// TIA Portal V21 export
FUNCTION_BLOCK "FB608"   // FB608, LAD
TITLE = FB608
{ S7_Optimized_Access := 'FALSE' }
AUTHOR : PRECISE
FAMILY : PRECISE
// CIP RECIRCULATION
// stored: AutoNumber false, SetENOAutomatically false
   VAR_INPUT
      CycleEnable : Bool;
      CycleRunning : Bool;
      SecPulse : Bool;
      AlwaysTrue : Bool;
      ActualTemperature : Real;
      ParaIn : "RecirculationInputs";
      ActualPressure : Real;
      ActualConductivity : Real;
   END_VAR
   VAR_OUTPUT
      Started : Bool;
      PressureUtilityValve : Bool;   // Air Utility
      AlkaliInValve : Bool;
      AlkaliPump : Bool;
      AcidInValve : Bool;
      AcidPump : Bool;
      "DosingValve(Cond)" : Bool;
      "DosingPump(Cond)" : Bool;
      HsbCmd : Bool;
      RecPump : Bool;
      ParaOut : "RecirculationOutputs";
      TimePv : DInt;
      StepStatus : String[60];
   END_VAR
   VAR_IN_OUT
      Over : Bool;
      OverTemp : Bool;
      ControlStarted : Bool;
      TimerPaused : Bool;
      PressurePostiveTol : Real;
      PressureNegativeTol : Real;
      LineValves : Bool;
      ActualRepetition : Int;
      SetTemperature { ExternalAccessible := 'False'; ExternalVisible := 'False'; ExternalWritable := 'False'} : Real;
      SetpH : Real;
      SetConductivity : Real;
      pHReached : Bool;
      ConductivityReached : Bool;
      CipSelected : Bool;
   END_VAR
   VAR
      ValveOnDelayPV : Int;
      ValveOffDelayPV : Int;
      ValveOnDelayPV_1 : Int;
      ValveOffDelayPV_1 : Int;
      ValveOnDelayPV_2 : Int;
      ValveOffDelayPV_2 : Int;
      TempPos : Real;
      RE1 : Bool;
      StepDelay { S7_SetPoint := 'True'} : "FB110";
      RE2 { S7_SetPoint := 'True'} : Bool;
      RE3 : Bool;
      RE4 : Bool;
      RE5 : Bool;
      Re6 : Bool;
      Re7 : Bool;
      "timer" : IEC_TIMER;
   END_VAR
   VAR_TEMP   // added for the SCL form of the ladder/FBD networks
      _w1 : Bool;
      _w2 : Bool;
   END_VAR
BEGIN

REGION Network 1: Logic for Output
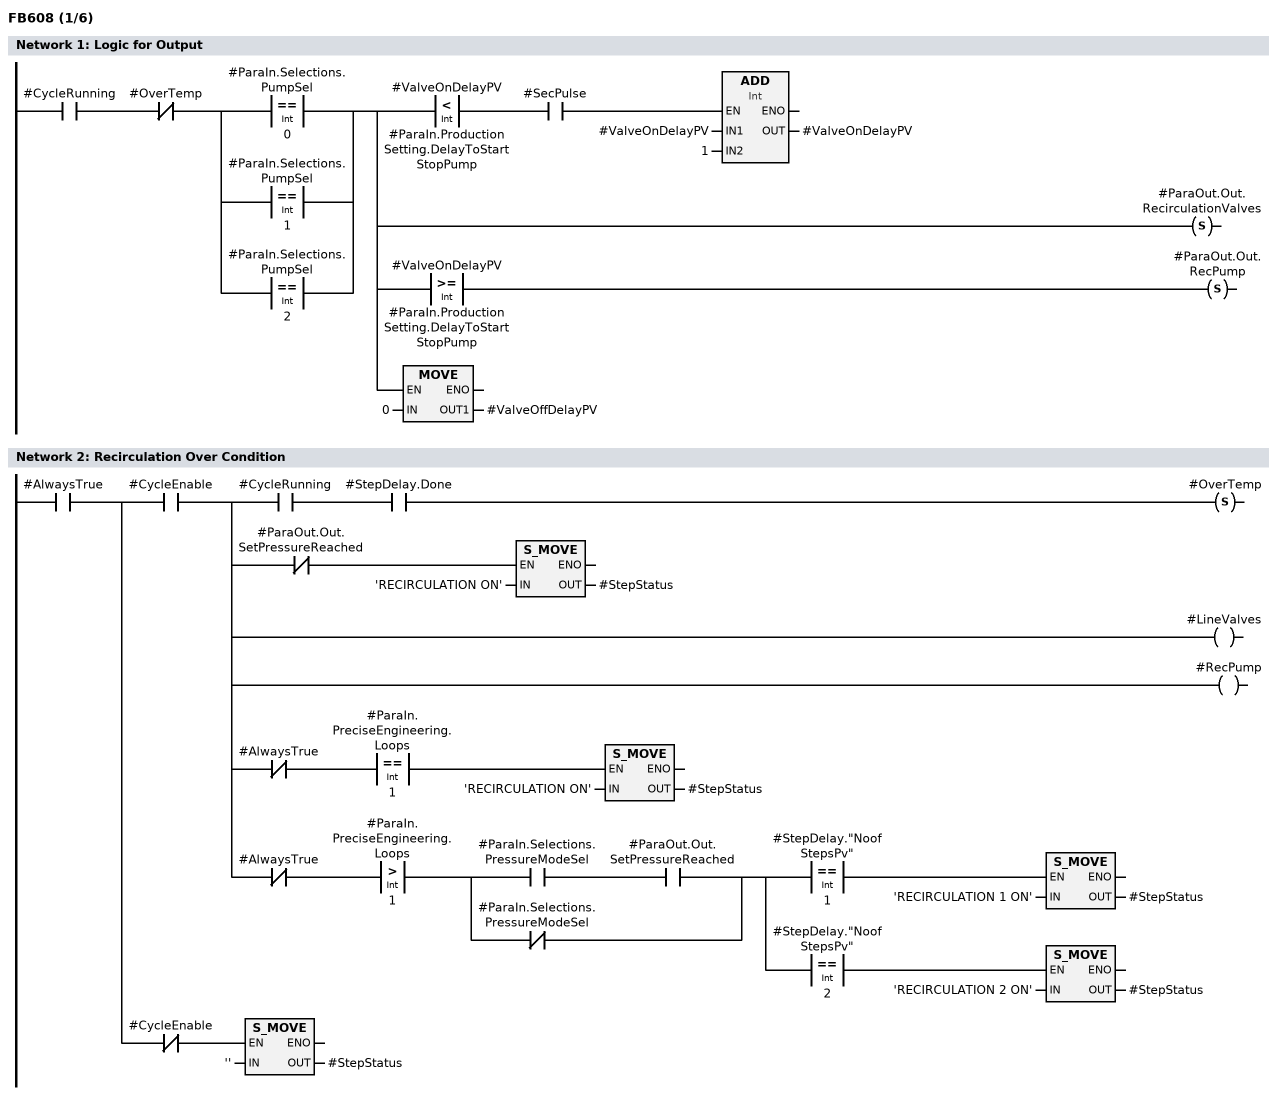
   RUNG wire#powerrail
      Contact( #CycleRunning )
      I_Contact( #OverTemp )
      wire#w1
      { S7_Templates := "SrcType := Int" } EQ_Contact(in1 := #ParaIn.Selections.PumpSel, in2 := 0)
      wire#w2
      { S7_Templates := "SrcType := Int" } LT_Contact(in1 := #ValveOnDelayPV, in2 := #ParaIn.ProductionSetting.DelayToStartStopPump)
      Contact( #SecPulse )
      { S7_Templates := "SrcType := Int"; S7_GenerateENO := "TRUE" } Add(in1 := #ValveOnDelayPV, in2 := 1, out => #ValveOnDelayPV)
   END_RUNG
   RUNG wire#w1
      { S7_Templates := "SrcType := Int" } EQ_Contact(in1 := #ParaIn.Selections.PumpSel, in2 := 1)
   END_RUNG wire#w2
   RUNG wire#w1
      { S7_Templates := "SrcType := Int" } EQ_Contact(in1 := #ParaIn.Selections.PumpSel, in2 := 2)
   END_RUNG wire#w2
   RUNG wire#w2
      S_Coil( #ParaOut.Out.RecirculationValves )
   END_RUNG
   RUNG wire#w2
      { S7_Templates := "SrcType := Int" } GE_Contact(in1 := #ValveOnDelayPV, in2 := #ParaIn.ProductionSetting.DelayToStartStopPump)
      S_Coil( #ParaOut.Out.RecPump )
   END_RUNG
   RUNG wire#w2
      { S7_GenerateENO := "TRUE" } Move(in := 0, out1 => #ValveOffDelayPV)
   END_RUNG
   // the same network as SCL:
   #_w1 := #CycleRunning AND NOT #OverTemp AND ((#ParaIn.Selections.PumpSel = 0) OR (#ParaIn.Selections.PumpSel = 1) OR (#ParaIn.Selections.PumpSel = 2));
   IF #_w1 AND (#ValveOnDelayPV < #ParaIn.ProductionSetting.DelayToStartStopPump) AND #SecPulse THEN
       #ValveOnDelayPV := #ValveOnDelayPV + 1;
   END_IF;
   IF #_w1 THEN #ParaOut.Out.RecirculationValves := TRUE; END_IF;
   IF #_w1 AND (#ValveOnDelayPV >= #ParaIn.ProductionSetting.DelayToStartStopPump) THEN
       #ParaOut.Out.RecPump := TRUE;
   END_IF;
   IF #_w1 THEN #ValveOffDelayPV := 0; END_IF;
END_REGION

REGION Network 2: Recirculation Over Condition
   RUNG wire#powerrail
      Contact( #AlwaysTrue )
      wire#w1
      Contact( #CycleEnable )
      wire#w2
      Contact( #CycleRunning )
      Contact( #StepDelay.Done )
      S_Coil( #OverTemp )
   END_RUNG
   RUNG wire#w2
      I_Contact( #ParaOut.Out.SetPressureReached )
      S_Move(in := 'RECIRCULATION ON', out => #StepStatus)
   END_RUNG
   RUNG wire#w2
      Coil( #LineValves )
   END_RUNG
   RUNG wire#w2
      Coil( #RecPump )
   END_RUNG
   RUNG wire#w2
      I_Contact( #AlwaysTrue )
      { S7_Templates := "SrcType := Int" } EQ_Contact(in1 := #ParaIn.PreciseEngineering.Loops, in2 := 1)
      S_Move(in := 'RECIRCULATION ON', out => #StepStatus)
   END_RUNG
   RUNG wire#w2
      I_Contact( #AlwaysTrue )
      { S7_Templates := "SrcType := Int" } GT_Contact(in1 := #ParaIn.PreciseEngineering.Loops, in2 := 1)
      wire#w3
      Contact( #ParaIn.Selections.PressureModeSel )
      Contact( #ParaOut.Out.SetPressureReached )
      wire#w4
      { S7_Templates := "SrcType := Int" } EQ_Contact(in1 := #StepDelay."Noof StepsPv", in2 := 1)
      S_Move(in := 'RECIRCULATION 1 ON', out => #StepStatus)
   END_RUNG
   RUNG wire#w3
      I_Contact( #ParaIn.Selections.PressureModeSel )
   END_RUNG wire#w4
   RUNG wire#w4
      { S7_Templates := "SrcType := Int" } EQ_Contact(in1 := #StepDelay."Noof StepsPv", in2 := 2)
      S_Move(in := 'RECIRCULATION 2 ON', out => #StepStatus)
   END_RUNG
   RUNG wire#w1
      I_Contact( #CycleEnable )
      S_Move(in := '', out => #StepStatus)
   END_RUNG
   // the same network as SCL:
   #_w1 := #AlwaysTrue AND #CycleEnable;
   IF #_w1 AND #CycleRunning AND #StepDelay.Done THEN #OverTemp := TRUE; END_IF;
   IF #_w1 AND NOT #ParaOut.Out.SetPressureReached THEN #StepStatus := 'RECIRCULATION ON'; END_IF;
   #LineValves := #_w1;
   #RecPump := #_w1;
   IF #_w1 AND NOT #AlwaysTrue AND (#ParaIn.PreciseEngineering.Loops = 1) THEN
       #StepStatus := 'RECIRCULATION ON';
   END_IF;
   #_w2 := #_w1 AND NOT #AlwaysTrue AND (#ParaIn.PreciseEngineering.Loops > 1) AND ((#ParaIn.Selections.PressureModeSel AND #ParaOut.Out.SetPressureReached) OR NOT #ParaIn.Selections.PressureModeSel);
   IF #_w2 AND (#StepDelay."Noof StepsPv" = 1) THEN #StepStatus := 'RECIRCULATION 1 ON'; END_IF;
   IF #_w2 AND (#StepDelay."Noof StepsPv" = 2) THEN #StepStatus := 'RECIRCULATION 2 ON'; END_IF;
   IF #AlwaysTrue AND NOT #CycleEnable THEN #StepStatus := ''; END_IF;
END_REGION

REGION Network 3: Recirculation Over
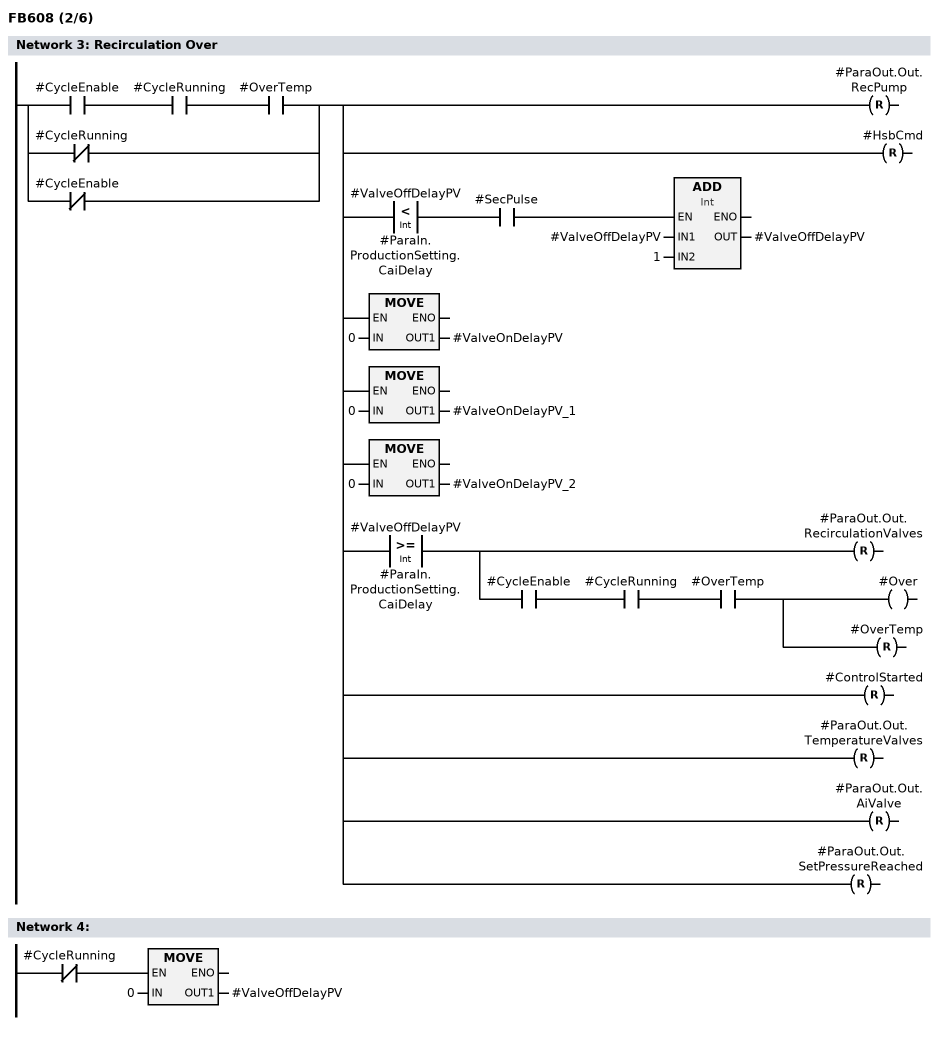
   RUNG wire#powerrail
      Contact( #CycleEnable )
      Contact( #CycleRunning )
      Contact( #OverTemp )
      wire#w1
      R_Coil( #ParaOut.Out.RecPump )
   END_RUNG
   RUNG wire#powerrail
      I_Contact( #CycleRunning )
   END_RUNG wire#w1
   RUNG wire#powerrail
      I_Contact( #CycleEnable )
   END_RUNG wire#w1
   RUNG wire#w1
      R_Coil( #HsbCmd )
   END_RUNG
   RUNG wire#w1
      { S7_Templates := "SrcType := Int" } LT_Contact(in1 := #ValveOffDelayPV, in2 := #ParaIn.ProductionSetting.CaiDelay)
      Contact( #SecPulse )
      { S7_Templates := "SrcType := Int"; S7_GenerateENO := "TRUE" } Add(in1 := #ValveOffDelayPV, in2 := 1, out => #ValveOffDelayPV)
   END_RUNG
   RUNG wire#w1
      { S7_GenerateENO := "TRUE" } Move(in := 0, out1 => #ValveOnDelayPV)
   END_RUNG
   RUNG wire#w1
      { S7_GenerateENO := "TRUE" } Move(in := 0, out1 => #ValveOnDelayPV_1)
   END_RUNG
   RUNG wire#w1
      { S7_GenerateENO := "TRUE" } Move(in := 0, out1 => #ValveOnDelayPV_2)
   END_RUNG
   RUNG wire#w1
      { S7_Templates := "SrcType := Int" } GE_Contact(in1 := #ValveOffDelayPV, in2 := #ParaIn.ProductionSetting.CaiDelay)
      wire#w2
      R_Coil( #ParaOut.Out.RecirculationValves )
   END_RUNG
   RUNG wire#w2
      Contact( #CycleEnable )
      Contact( #CycleRunning )
      Contact( #OverTemp )
      wire#w3
      Coil( #Over )
   END_RUNG
   RUNG wire#w3
      R_Coil( #OverTemp )
   END_RUNG
   RUNG wire#w1
      R_Coil( #ControlStarted )
   END_RUNG
   RUNG wire#w1
      R_Coil( #ParaOut.Out.TemperatureValves )
   END_RUNG
   RUNG wire#w1
      R_Coil( #ParaOut.Out.AiValve )
   END_RUNG
   RUNG wire#w1
      R_Coil( #ParaOut.Out.SetPressureReached )
   END_RUNG
   // the same network as SCL:
   #_w1 := (#CycleEnable AND #CycleRunning AND #OverTemp) OR NOT #CycleRunning OR NOT #CycleEnable;
   IF #_w1 THEN
       #ParaOut.Out.RecPump := FALSE;
       #HsbCmd := FALSE;
   END_IF;
   IF #_w1 AND (#ValveOffDelayPV < #ParaIn.ProductionSetting.CaiDelay) AND #SecPulse THEN
       #ValveOffDelayPV := #ValveOffDelayPV + 1;
   END_IF;
   IF #_w1 THEN
       #ValveOnDelayPV := 0;
       #ValveOnDelayPV_1 := 0;
       #ValveOnDelayPV_2 := 0;
   END_IF;
   #_w2 := #_w1 AND (#ValveOffDelayPV >= #ParaIn.ProductionSetting.CaiDelay);
   IF #_w2 THEN #ParaOut.Out.RecirculationValves := FALSE; END_IF;
   #Over := #_w2 AND #CycleEnable AND #CycleRunning AND #OverTemp;
   IF #Over THEN #OverTemp := FALSE; END_IF;
   IF #_w1 THEN
       #ControlStarted := FALSE;
       #ParaOut.Out.TemperatureValves := FALSE;
       #ParaOut.Out.AiValve := FALSE;
       #ParaOut.Out.SetPressureReached := FALSE;
   END_IF;
END_REGION

REGION Network 4
   RUNG wire#powerrail
      I_Contact( #CycleRunning )
      Move(in := 0, out1 => #ValveOffDelayPV)
   END_RUNG
   // the same network as SCL:
   IF NOT #CycleRunning THEN #ValveOffDelayPV := 0; END_IF;
END_REGION

REGION Network 5: StepDelay.StepTimeSV
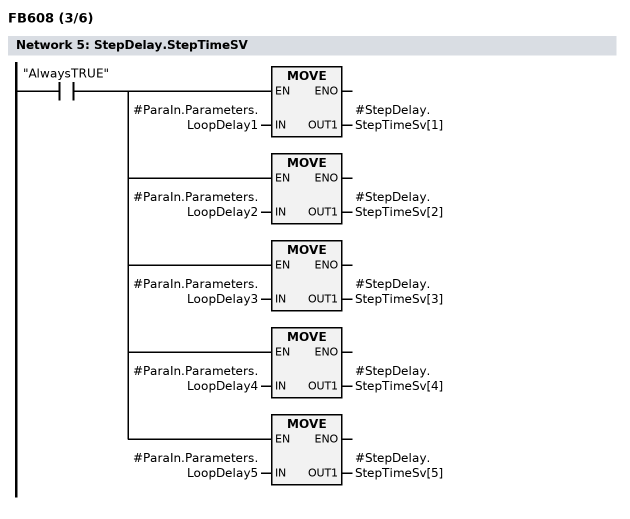
   RUNG wire#powerrail
      Contact( "AlwaysTRUE" )
      wire#w1
      Move(in := #ParaIn.Parameters.LoopDelay1, out1 => #StepDelay.StepTimeSv[1])
   END_RUNG
   RUNG wire#w1
      Move(in := #ParaIn.Parameters.LoopDelay2, out1 => #StepDelay.StepTimeSv[2])
   END_RUNG
   RUNG wire#w1
      Move(in := #ParaIn.Parameters.LoopDelay3, out1 => #StepDelay.StepTimeSv[3])
   END_RUNG
   RUNG wire#w1
      Move(in := #ParaIn.Parameters.LoopDelay4, out1 => #StepDelay.StepTimeSv[4])
   END_RUNG
   RUNG wire#w1
      Move(in := #ParaIn.Parameters.LoopDelay5, out1 => #StepDelay.StepTimeSv[5])
   END_RUNG
   // the same network as SCL:
   IF "AlwaysTRUE" THEN
       #StepDelay.StepTimeSv[1] := #ParaIn.Parameters.LoopDelay1;
       #StepDelay.StepTimeSv[2] := #ParaIn.Parameters.LoopDelay2;
       #StepDelay.StepTimeSv[3] := #ParaIn.Parameters.LoopDelay3;
       #StepDelay.StepTimeSv[4] := #ParaIn.Parameters.LoopDelay4;
       #StepDelay.StepTimeSv[5] := #ParaIn.Parameters.LoopDelay5;
   END_IF;
END_REGION

REGION Network 6: sv and pv for run screen
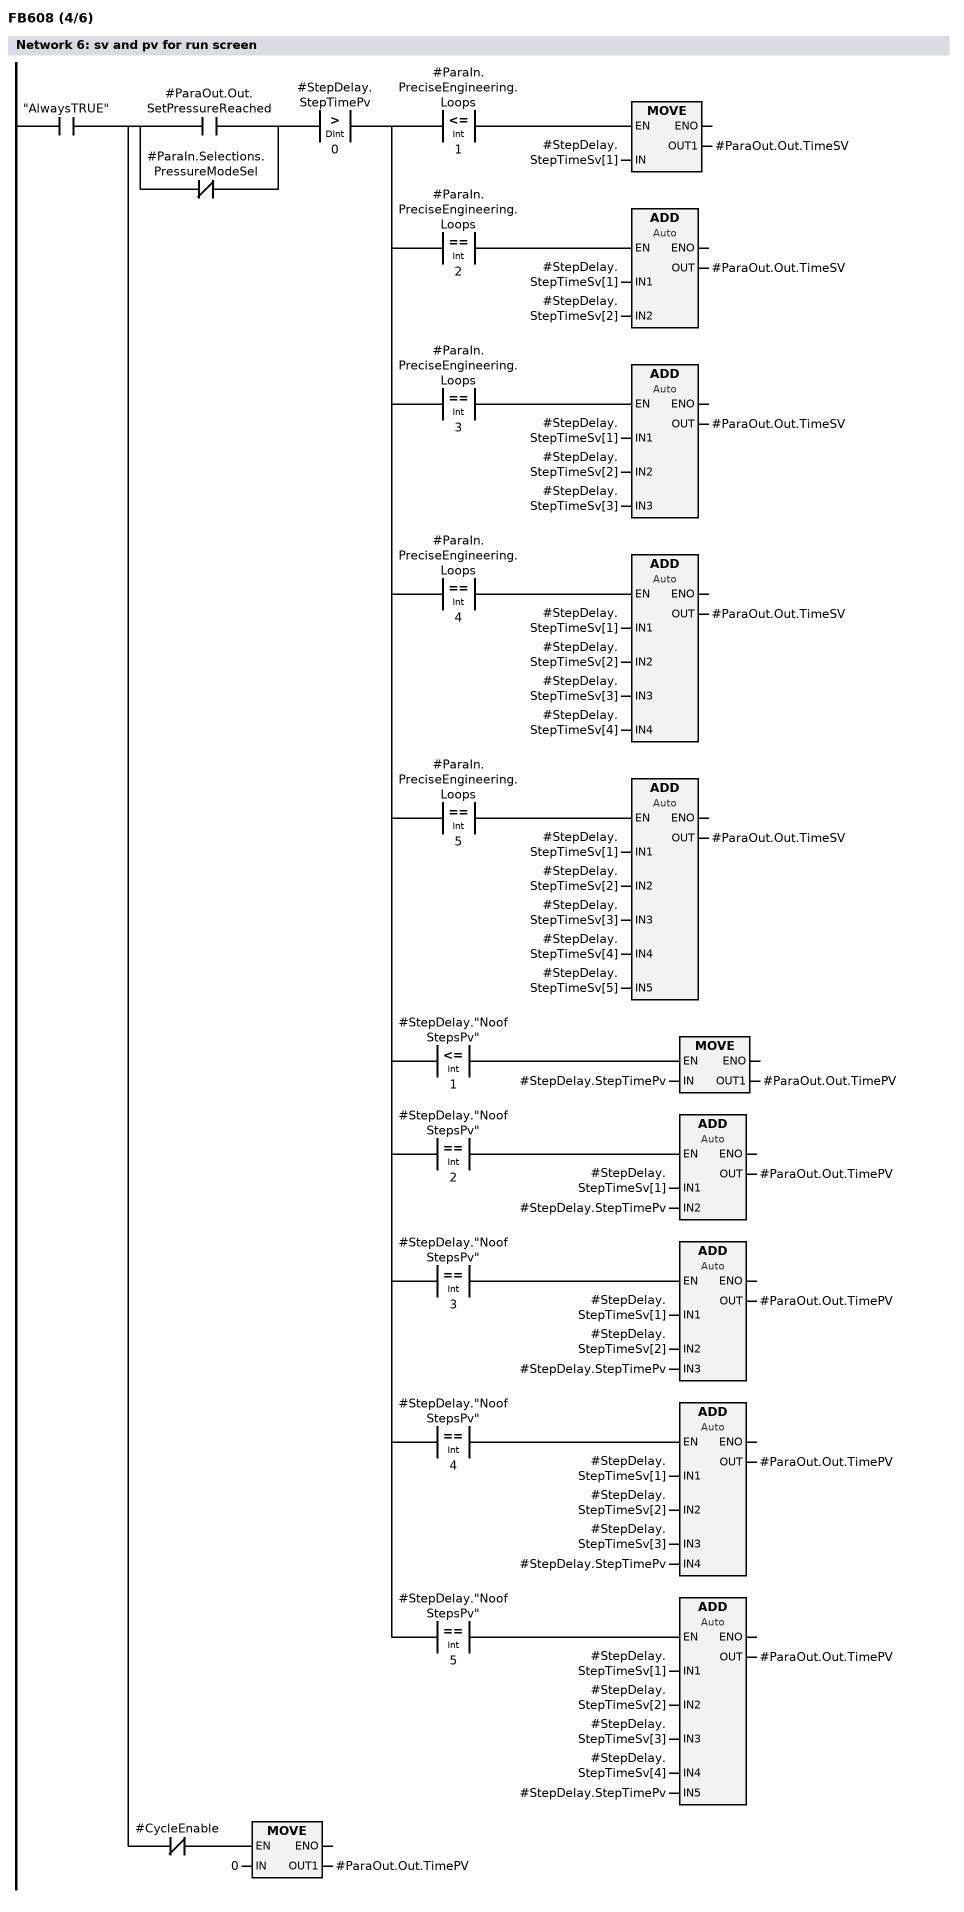
   RUNG wire#powerrail
      Contact( "AlwaysTRUE" )
      wire#w1
      Contact( #ParaOut.Out.SetPressureReached )
      wire#w2
      { S7_Templates := "SrcType := DInt" } GT_Contact(in1 := #StepDelay.StepTimePv, in2 := 0)
      wire#w3
      { S7_Templates := "SrcType := Int" } LE_Contact(in1 := #ParaIn.PreciseEngineering.Loops, in2 := 1)
      Move(in := #StepDelay.StepTimeSv[1], out1 => #ParaOut.Out.TimeSV)
   END_RUNG
   RUNG wire#w1
      I_Contact( #ParaIn.Selections.PressureModeSel )
   END_RUNG wire#w2
   RUNG wire#w3
      { S7_Templates := "SrcType := Int" } EQ_Contact(in1 := #ParaIn.PreciseEngineering.Loops, in2 := 2)
      Add(in1 := #StepDelay.StepTimeSv[1], in2 := #StepDelay.StepTimeSv[2], out => #ParaOut.Out.TimeSV)
   END_RUNG
   RUNG wire#w3
      { S7_Templates := "SrcType := Int" } EQ_Contact(in1 := #ParaIn.PreciseEngineering.Loops, in2 := 3)
      Add(in1 := #StepDelay.StepTimeSv[1], in2 := #StepDelay.StepTimeSv[2], in3 := #StepDelay.StepTimeSv[3], out => #ParaOut.Out.TimeSV)
   END_RUNG
   RUNG wire#w3
      { S7_Templates := "SrcType := Int" } EQ_Contact(in1 := #ParaIn.PreciseEngineering.Loops, in2 := 4)
      Add(in1 := #StepDelay.StepTimeSv[1], in2 := #StepDelay.StepTimeSv[2], in3 := #StepDelay.StepTimeSv[3], in4 := #StepDelay.StepTimeSv[4], out => #ParaOut.Out.TimeSV)
   END_RUNG
   RUNG wire#w3
      { S7_Templates := "SrcType := Int" } EQ_Contact(in1 := #ParaIn.PreciseEngineering.Loops, in2 := 5)
      Add(in1 := #StepDelay.StepTimeSv[1], in2 := #StepDelay.StepTimeSv[2], in3 := #StepDelay.StepTimeSv[3], in4 := #StepDelay.StepTimeSv[4], in5 := #StepDelay.StepTimeSv[5], out => #ParaOut.Out.TimeSV)
   END_RUNG
   RUNG wire#w3
      { S7_Templates := "SrcType := Int" } LE_Contact(in1 := #StepDelay."Noof StepsPv", in2 := 1)
      Move(in := #StepDelay.StepTimePv, out1 => #ParaOut.Out.TimePV)
   END_RUNG
   RUNG wire#w3
      { S7_Templates := "SrcType := Int" } EQ_Contact(in1 := #StepDelay."Noof StepsPv", in2 := 2)
      Add(in1 := #StepDelay.StepTimeSv[1], in2 := #StepDelay.StepTimePv, out => #ParaOut.Out.TimePV)
   END_RUNG
   RUNG wire#w3
      { S7_Templates := "SrcType := Int" } EQ_Contact(in1 := #StepDelay."Noof StepsPv", in2 := 3)
      Add(in1 := #StepDelay.StepTimeSv[1], in2 := #StepDelay.StepTimeSv[2], in3 := #StepDelay.StepTimePv, out => #ParaOut.Out.TimePV)
   END_RUNG
   RUNG wire#w3
      { S7_Templates := "SrcType := Int" } EQ_Contact(in1 := #StepDelay."Noof StepsPv", in2 := 4)
      Add(in1 := #StepDelay.StepTimeSv[1], in2 := #StepDelay.StepTimeSv[2], in3 := #StepDelay.StepTimeSv[3], in4 := #StepDelay.StepTimePv, out => #ParaOut.Out.TimePV)
   END_RUNG
   RUNG wire#w3
      { S7_Templates := "SrcType := Int" } EQ_Contact(in1 := #StepDelay."Noof StepsPv", in2 := 5)
      Add(in1 := #StepDelay.StepTimeSv[1], in2 := #StepDelay.StepTimeSv[2], in3 := #StepDelay.StepTimeSv[3], in4 := #StepDelay.StepTimeSv[4], in5 := #StepDelay.StepTimePv, out => #ParaOut.Out.TimePV)
   END_RUNG
   RUNG wire#w1
      I_Contact( #CycleEnable )
      Move(in := 0, out1 => #ParaOut.Out.TimePV)
   END_RUNG
   // the same network as SCL:
   #_w1 := "AlwaysTRUE" AND (#ParaOut.Out.SetPressureReached OR NOT #ParaIn.Selections.PressureModeSel) AND (#StepDelay.StepTimePv > 0);
   IF #_w1 AND (#ParaIn.PreciseEngineering.Loops <= 1) THEN
       #ParaOut.Out.TimeSV := #StepDelay.StepTimeSv[1];
   END_IF;
   IF #_w1 AND (#ParaIn.PreciseEngineering.Loops = 2) THEN
       #ParaOut.Out.TimeSV := #StepDelay.StepTimeSv[1] + #StepDelay.StepTimeSv[2];
   END_IF;
   IF #_w1 AND (#ParaIn.PreciseEngineering.Loops = 3) THEN
       #ParaOut.Out.TimeSV := #StepDelay.StepTimeSv[1] + #StepDelay.StepTimeSv[2] + #StepDelay.StepTimeSv[3];
   END_IF;
   IF #_w1 AND (#ParaIn.PreciseEngineering.Loops = 4) THEN
       #ParaOut.Out.TimeSV := #StepDelay.StepTimeSv[1] + #StepDelay.StepTimeSv[2] + #StepDelay.StepTimeSv[3] + #StepDelay.StepTimeSv[4];
   END_IF;
   IF #_w1 AND (#ParaIn.PreciseEngineering.Loops = 5) THEN
       #ParaOut.Out.TimeSV := #StepDelay.StepTimeSv[1] + #StepDelay.StepTimeSv[2] + #StepDelay.StepTimeSv[3] + #StepDelay.StepTimeSv[4] + #StepDelay.StepTimeSv[5];
   END_IF;
   IF #_w1 AND (#StepDelay."Noof StepsPv" <= 1) THEN #ParaOut.Out.TimePV := #StepDelay.StepTimePv; END_IF;
   IF #_w1 AND (#StepDelay."Noof StepsPv" = 2) THEN
       #ParaOut.Out.TimePV := #StepDelay.StepTimeSv[1] + #StepDelay.StepTimePv;
   END_IF;
   IF #_w1 AND (#StepDelay."Noof StepsPv" = 3) THEN
       #ParaOut.Out.TimePV := #StepDelay.StepTimeSv[1] + #StepDelay.StepTimeSv[2] + #StepDelay.StepTimePv;
   END_IF;
   IF #_w1 AND (#StepDelay."Noof StepsPv" = 4) THEN
       #ParaOut.Out.TimePV := #StepDelay.StepTimeSv[1] + #StepDelay.StepTimeSv[2] + #StepDelay.StepTimeSv[3] + #StepDelay.StepTimePv;
   END_IF;
   IF #_w1 AND (#StepDelay."Noof StepsPv" = 5) THEN
       #ParaOut.Out.TimePV := #StepDelay.StepTimeSv[1] + #StepDelay.StepTimeSv[2] + #StepDelay.StepTimeSv[3] + #StepDelay.StepTimeSv[4] + #StepDelay.StepTimePv;
   END_IF;
   IF "AlwaysTRUE" AND NOT #CycleEnable THEN #ParaOut.Out.TimePV := 0; END_IF;
END_REGION

REGION Network 7: #StepDelay
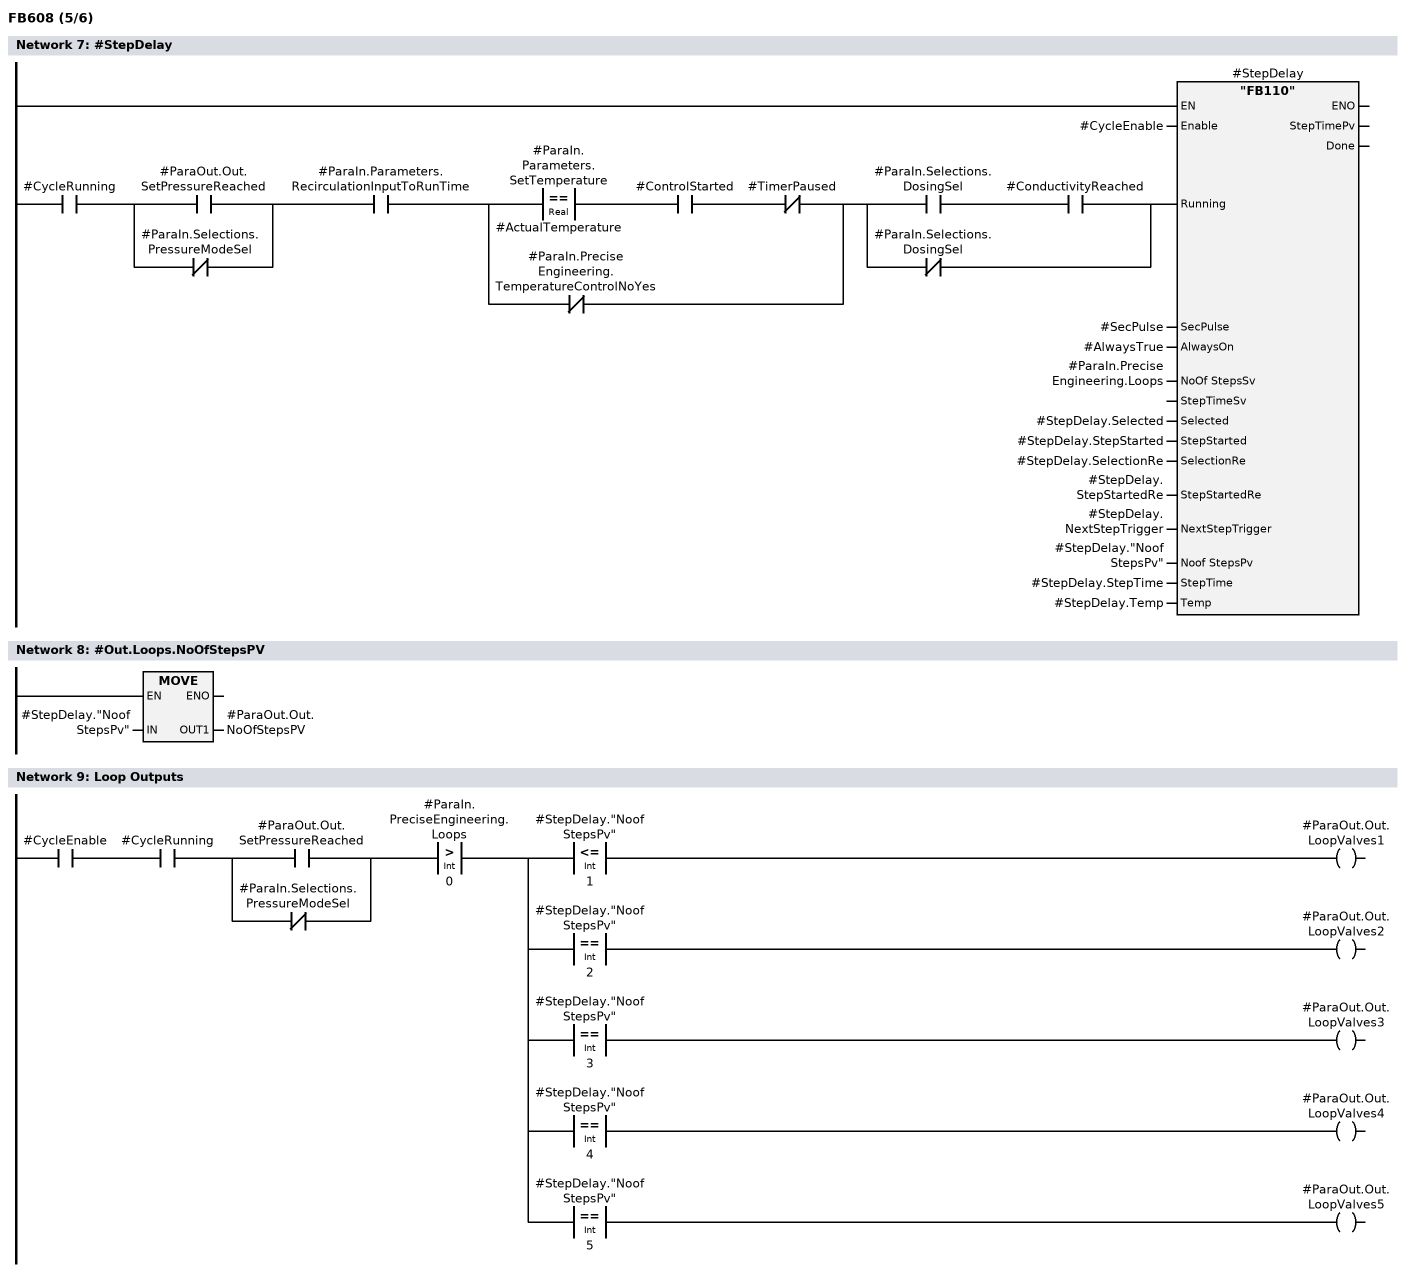
   RUNG wire#powerrail
      #StepDelay(Running := wire#w5, Enable := #CycleEnable, SecPulse := #SecPulse, AlwaysOn := #AlwaysTrue, "NoOf StepsSv" := #ParaIn.PreciseEngineering.Loops, StepTimeSv :=, Selected := #StepDelay.Selected, StepStarted := #StepDelay.StepStarted, SelectionRe := #StepDelay.SelectionRe, StepStartedRe := #StepDelay.StepStartedRe, NextStepTrigger := #StepDelay.NextStepTrigger, "Noof StepsPv" := #StepDelay."Noof StepsPv", StepTime := #StepDelay.StepTime, Temp := #StepDelay.Temp, StepTimePv =>, Done =>)
   END_RUNG
   RUNG wire#powerrail
      Contact( #CycleRunning )
      wire#w1
      Contact( #ParaOut.Out.SetPressureReached )
      wire#w2
      Contact( #ParaIn.Parameters.RecirculationInputToRunTime )
      wire#w3
      { S7_Templates := "SrcType := Real" } EQ_Contact(in1 := #ParaIn.Parameters.SetTemperature, in2 := #ActualTemperature)
      Contact( #ControlStarted )
      I_Contact( #TimerPaused )
      wire#w4
      Contact( #ParaIn.Selections.DosingSel )
      Contact( #ConductivityReached )
   END_RUNG wire#w5
   RUNG wire#w1
      I_Contact( #ParaIn.Selections.PressureModeSel )
   END_RUNG wire#w2
   RUNG wire#w3
      I_Contact( #ParaIn.PreciseEngineering.TemperatureControlNoYes )
   END_RUNG wire#w4
   RUNG wire#w4
      I_Contact( #ParaIn.Selections.DosingSel )
   END_RUNG wire#w5
   // the same network as SCL:
   #StepDelay(Enable := #CycleEnable,   // "FB110"
              Running := #CycleRunning AND (#ParaOut.Out.SetPressureReached OR NOT #ParaIn.Selections.PressureModeSel) AND #ParaIn.Parameters.RecirculationInputToRunTime AND (((#ParaIn.Parameters.SetTemperature = #ActualTemperature) AND #ControlStarted AND NOT #TimerPaused) OR NOT #ParaIn.PreciseEngineering.TemperatureControlNoYes) AND ((#ParaIn.Selections.DosingSel AND #ConductivityReached) OR NOT #ParaIn.Selections.DosingSel),
              SecPulse := #SecPulse,
              AlwaysOn := #AlwaysTrue,
              "NoOf StepsSv" := #ParaIn.PreciseEngineering.Loops,
              Selected := #StepDelay.Selected,
              StepStarted := #StepDelay.StepStarted,
              SelectionRe := #StepDelay.SelectionRe,
              StepStartedRe := #StepDelay.StepStartedRe,
              NextStepTrigger := #StepDelay.NextStepTrigger,
              "Noof StepsPv" := #StepDelay."Noof StepsPv",
              StepTime := #StepDelay.StepTime,
              Temp := #StepDelay.Temp);
END_REGION

REGION Network 8: #Out.Loops.NoOfStepsPV
   RUNG wire#powerrail
      Move(in := #StepDelay."Noof StepsPv", out1 => #ParaOut.Out.NoOfStepsPV)
   END_RUNG
   // the same network as SCL:
   #ParaOut.Out.NoOfStepsPV := #StepDelay."Noof StepsPv";
END_REGION

REGION Network 9: Loop Outputs
   RUNG wire#powerrail
      Contact( #CycleEnable )
      Contact( #CycleRunning )
      wire#w1
      Contact( #ParaOut.Out.SetPressureReached )
      wire#w2
      { S7_Templates := "SrcType := Int" } GT_Contact(in1 := #ParaIn.PreciseEngineering.Loops, in2 := 0)
      wire#w3
      { S7_Templates := "SrcType := Int" } LE_Contact(in1 := #StepDelay."Noof StepsPv", in2 := 1)
      Coil( #ParaOut.Out.LoopValves1 )
   END_RUNG
   RUNG wire#w1
      I_Contact( #ParaIn.Selections.PressureModeSel )
   END_RUNG wire#w2
   RUNG wire#w3
      { S7_Templates := "SrcType := Int" } EQ_Contact(in1 := #StepDelay."Noof StepsPv", in2 := 2)
      Coil( #ParaOut.Out.LoopValves2 )
   END_RUNG
   RUNG wire#w3
      { S7_Templates := "SrcType := Int" } EQ_Contact(in1 := #StepDelay."Noof StepsPv", in2 := 3)
      Coil( #ParaOut.Out.LoopValves3 )
   END_RUNG
   RUNG wire#w3
      { S7_Templates := "SrcType := Int" } EQ_Contact(in1 := #StepDelay."Noof StepsPv", in2 := 4)
      Coil( #ParaOut.Out.LoopValves4 )
   END_RUNG
   RUNG wire#w3
      { S7_Templates := "SrcType := Int" } EQ_Contact(in1 := #StepDelay."Noof StepsPv", in2 := 5)
      Coil( #ParaOut.Out.LoopValves5 )
   END_RUNG
   // the same network as SCL:
   #_w1 := #CycleEnable AND #CycleRunning AND (#ParaOut.Out.SetPressureReached OR NOT #ParaIn.Selections.PressureModeSel) AND (#ParaIn.PreciseEngineering.Loops > 0);
   #ParaOut.Out.LoopValves1 := #_w1 AND (#StepDelay."Noof StepsPv" <= 1);
   #ParaOut.Out.LoopValves2 := #_w1 AND (#StepDelay."Noof StepsPv" = 2);
   #ParaOut.Out.LoopValves3 := #_w1 AND (#StepDelay."Noof StepsPv" = 3);
   #ParaOut.Out.LoopValves4 := #_w1 AND (#StepDelay."Noof StepsPv" = 4);
   #ParaOut.Out.LoopValves5 := #_w1 AND (#StepDelay."Noof StepsPv" = 5);
END_REGION

REGION Network 10: Reset
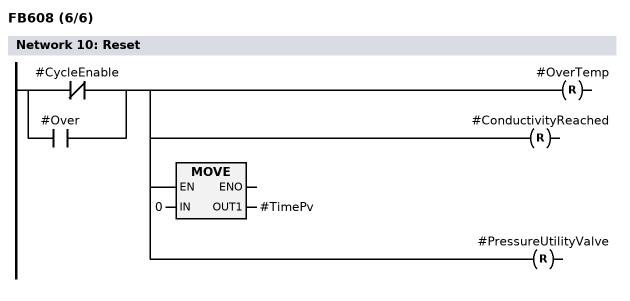
   RUNG wire#powerrail
      I_Contact( #CycleEnable )
      wire#w1
      R_Coil( #OverTemp )
   END_RUNG
   RUNG wire#powerrail
      Contact( #Over )
   END_RUNG wire#w1
   RUNG wire#w1
      R_Coil( #ConductivityReached )
   END_RUNG
   RUNG wire#w1
      { S7_GenerateENO := "TRUE" } Move(in := 0, out1 => #TimePv)
   END_RUNG
   RUNG wire#w1
      R_Coil( #PressureUtilityValve )
   END_RUNG
   // the same network as SCL:
   IF NOT #CycleEnable OR #Over THEN
       #OverTemp := FALSE;
       #ConductivityReached := FALSE;
       #TimePv := 0;
       #PressureUtilityValve := FALSE;
   END_IF;
END_REGION
END_FUNCTION_BLOCK
